INTERFACE IMachine

PROPERTY PMLState : PackMLState
GET
END_GET
END_PROPERTY

END_INTERFACE

(* stored: Version 1.1.0.1, ProductVersion 3.1.4024.9
   Itf IMachine: Id {2f2a2bb8-28a0-4228-9323-58e2c8d4e0dc}
   Property PMLState: Id {ca082088-8442-42b0-bf5a-85ad1b42830d}
   Get Get: Id {42dbe94e-961d-4466-bac8-ac3c6c5ba5b7} *)
